TYPE E_GantryMode :
(
    GantryModeCoupled := 0,
    GantryModeDecoupled	:= 1
);
END_TYPE

(* stored: Version 1.1.0.1, ProductVersion 3.1.4020.12
   DUT E_GantryMode: Id {d4415ee5-967f-4ffb-be4f-02092fdb80c5} *)
